Universal Robots PolyScope program: robot_control_25.urp

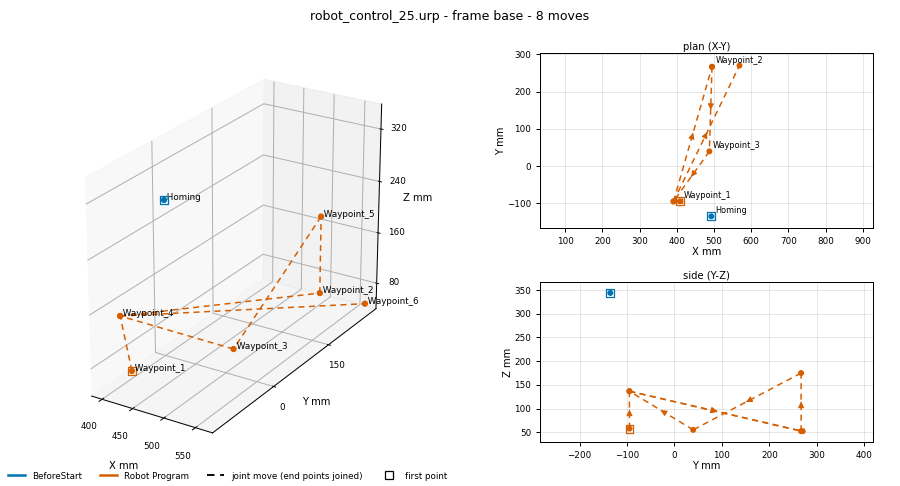
[picture p0: tool path of robot_control_25.urp in frame base, 8 of 8 moves have a stored position in this frame; points joined in program order, loops and branches not executed]
Program robot_control_25 (installation=tangram_inst directory=/programs/usbdisk/new folder createdIn=5.14.5 lastSavedIn=5.14.5 robotSerialNumber=20225501312)
Calibrated DH parameters: a=[0.000177, -0.405867, -0.359302, -0.000009, 0.00008, 0]; d=[0.162556, -59.259033, 22.634856, 36.757695, 0.099775, 0.099535]; alpha=[1.570983, 0.00214, 0.004319, 1.570342, -1.569638, 0]; deltaTheta=[0, -0.302866, 6.171309, 0.414749, 0.000002, -0.000001]
InitVariablesNode
BeforeStart
  MoveJ speed 60 deg/s, acceleration 80 deg/s^2 (useActiveTCP=true) feature=Base
    Waypoint Homing: TCP in base x=492.783 y=-135.148 z=343.84 mm, rx=2.219 ry=-2.2206 rz=0.0062 rad; joints [0.001, -89.999, -90, -89.999, 90, -0.001] deg; TCP offset x=0 y=0 z=145 mm, rx=0 ry=0 rz=0 rad
    URCap Gripper Activate (Robotiq_Grippers, Robotiq Inc.) dataModel(ResetAndActivateKey=true)
    URCap Gripper (Robotiq_Grippers, Robotiq Inc.) dataModel(position=0.0, force=100.0, speed=100.0, positionInDouble=0.0, forceInDouble=100.0, speedInDouble=100.0, slaveIds=[2], blocking=true, robotCompliant=false)
Robot Program (runOnlyOnce=true)
  MoveJ speed 60 deg/s, acceleration 80 deg/s^2 (useActiveTCP=true) feature=Base
    Waypoint Waypoint_1: TCP in base x=408.294 y=-94.649 z=57.984 mm, rx=2.2191 ry=-2.2206 rz=0.0062 rad; joints [5.712, -94.192, -133.286, -42.543, 89.856, 5.846] deg; TCP offset x=0 y=0 z=140 mm, rx=0 ry=0 rz=0 rad
    URCap Gripper (Robotiq_Grippers, Robotiq Inc.) dataModel(position=100.0, force=100.0, speed=100.0, positionInDouble=100.0, forceInDouble=100.0, speedInDouble=100.0, slaveIds=[2], blocking=true, robotCompliant=false)
    Waypoint Waypoint_4: TCP in base x=391.131 y=-94.961 z=136.797 mm, rx=2.2191 ry=-2.2206 rz=0.0062 rad; joints [5.938, -82.721, -129.328, -57.974, 89.893, 6.036] deg
  MoveJ speed 60 deg/s, acceleration 80 deg/s^2 (useActiveTCP=true) feature=Base
    Waypoint Waypoint_2: TCP in base x=494.616 y=266.887 z=52.512 mm, rx=2.2191 ry=-2.2206 rz=0.0062 rad; joints [42.228, -111.173, -110.71, -48.301, 89.934, 42.372] deg; TCP offset x=0 y=0 z=145 mm, rx=0 ry=0 rz=0 rad
    URCap Gripper (Robotiq_Grippers, Robotiq Inc.) dataModel(position=0.0, force=100.0, speed=100.0, positionInDouble=0.0, forceInDouble=100.0, speedInDouble=100.0, slaveIds=[2], blocking=true, robotCompliant=false)
    Waypoint Waypoint_5: TCP in base x=494.616 y=266.874 z=175.058 mm, rx=2.2191 ry=-2.2206 rz=0.0062 rad; joints [42.236, -102.11, -102.565, -65.508, 89.981, 42.327] deg; TCP offset x=0 y=0 z=140 mm, rx=0 ry=0 rz=0 rad
  MoveJ speed 60 deg/s, acceleration 80 deg/s^2 (useActiveTCP=true) feature=Base
    Waypoint Waypoint_3: TCP in base x=487.539 y=39.493 z=55.364 mm, rx=2.2189 ry=-2.2206 rz=0.0061 rad; joints [20.636, -103.157, -122.728, -44.214, 89.878, 20.78] deg
    URCap Gripper (Robotiq_Grippers, Robotiq Inc.) dataModel(position=100.0, force=100.0, speed=100.0, positionInDouble=100.0, forceInDouble=100.0, speedInDouble=100.0, slaveIds=[2], blocking=true, robotCompliant=false)
    Waypoint Waypoint_4: TCP in base x=391.131 y=-94.961 z=136.797 mm, rx=2.2191 ry=-2.2206 rz=0.0062 rad; joints [5.938, -82.721, -129.328, -57.974, 89.893, 6.036] deg
  MoveJ speed 60 deg/s, acceleration 80 deg/s^2 (useActiveTCP=true) feature=Base
    Waypoint Waypoint_6: TCP in base x=568.49 y=270.258 z=52.511 mm, rx=2.2191 ry=-2.2206 rz=0.0063 rad; joints [37.792, -119.02, -99.13, -52.017, 89.952, 37.939] deg
    URCap Gripper (Robotiq_Grippers, Robotiq Inc.) dataModel(position=0.0, force=100.0, speed=100.0, positionInDouble=0.0, forceInDouble=100.0, speedInDouble=100.0, slaveIds=[2], blocking=true, robotCompliant=false)
